(* IEC 61131-3 sources: RetroPLC_IDE/RetroPLC.Shell/ProjectFiles/POUs/Programs, 2 files *)

(* ---- Blink.st ---- *)
PROGRAM Blink
VAR
    timer : TON;
    runLamp AT %QX0.1 : BOOL;
END_VAR

timer(IN := NOT timer.Q, PT := T#500ms);

IF timer.Q THEN
    runLamp := NOT runLamp;
END_IF;
END_PROGRAM

(* ---- Main.st ---- *)
PROGRAM Main
VAR
    motor : MotorController;
    startButton AT %IX0.0 : BOOL;
    stopButton AT %IX0.1 : BOOL;
    motorEnable AT %QX0.0 : BOOL;
END_VAR

motor(
    StartRequest := startButton,
    StopRequest := stopButton
);

motorEnable := motor.IsRunning;
END_PROGRAM
